// TIA Portal V17 export
// export: Created 2025-03-07T09:17:44.8534748Z, ExportSetting WithDefaults, DisplayName Totally Integrated Automation Portal, DisplayVersion V17 Update 8, DisplayName TIA Portal Openness, DisplayVersion V17 Update 8, DisplayName TIA Portal Version Control Interface, DisplayVersion V17, DisplayName SINAMICS Startdrive Advanced, DisplayVersion V17 SP2, DisplayName SINAMICS Startdrive G110M, G120, G120C, G120D, G120P, G115D, DisplayVersion V17 SP2, DisplayName SINAMICS Startdrive G130, G150, S120, S150, SINAMICS MV, S210, DisplayVersion V17 SP2, DisplayName STEP 7 Professional, DisplayVersion V17 Update 8, DisplayName SINUMERIK ONE STEP 7 Toolbox, DisplayVersion V17 Update 12, DisplayName SINUMERIK 840D sl STEP 7 Toolbox, DisplayVersion V17 Update 12, DisplayName STEP 7 Safety, DisplayVersion V17 Update 6, DisplayName WinCC Advanced, DisplayVersion V17 Update 8
DATA_BLOCK "DB2002_BA_MODES_MG1"   // DB2002
{ DB_Accessible_From_OPC_UA := 'FALSE' }
VERSION : 0.1
// stored: AutoNumber false, DBAccessibleFromOPCUA false, DBAccessibleFromWebserver true, InstanceOfName FB2002_BA_MODE, InstanceOfType FB
"FB2002_BA_MODE"
   // VAR_INPUT
   //    OPTIONS_0 { ExternalAccessible := 'False'; ExternalVisible := 'False'; ExternalWritable := 'False'} : Byte;
   //    BA1_BUTTON_I { ExternalAccessible := 'False'; ExternalVisible := 'False'; ExternalWritable := 'False'} : Bool;
   //    BA2_BUTTON_I { ExternalAccessible := 'False'; ExternalVisible := 'False'; ExternalWritable := 'False'} : Bool;
   //    BA3_BUTTON_I { ExternalAccessible := 'False'; ExternalVisible := 'False'; ExternalWritable := 'False'} : Bool;
   //    BA5_BUTTON_I { ExternalAccessible := 'False'; ExternalVisible := 'False'; ExternalWritable := 'False'} : Bool;
   //    SAFETY_ENABLED_W_DOOR_OPENED { ExternalAccessible := 'False'; ExternalVisible := 'False'; ExternalWritable := 'False'} : Bool;
   //    SAFETY_GATES_CLSD_AND_LCKD { ExternalAccessible := 'False'; ExternalVisible := 'False'; ExternalWritable := 'False'} : Bool;
   //    START_SERVICES_GLOBAL { ExternalAccessible := 'False'; ExternalVisible := 'False'; ExternalWritable := 'False'} : Bool;
   //    ANY_MCH_CYCLE_RUN { ExternalAccessible := 'False'; ExternalVisible := 'False'; ExternalWritable := 'False'} : Bool;
   //    MCH_RESET_FAULTS { ExternalAccessible := 'False'; ExternalVisible := 'False'; ExternalWritable := 'False'} : Bool;
   // END_VAR
   // VAR_OUTPUT
   //    NO_BA_MODE_SLCTD_WRN { ExternalAccessible := 'False'; ExternalVisible := 'False'; ExternalWritable := 'False'} : Bool;
   //    CHANGE_TO_BA1_MODE_WRN { ExternalAccessible := 'False'; ExternalVisible := 'False'; ExternalWritable := 'False'} : Bool;
   //    CHANGE_TO_BA2_MODE_WRN { ExternalAccessible := 'False'; ExternalVisible := 'False'; ExternalWritable := 'False'} : Bool;
   //    CHANGE_TO_BA3_MODE_WRN { ExternalAccessible := 'False'; ExternalVisible := 'False'; ExternalWritable := 'False'} : Bool;
   //    CHANGE_TO_BA5_MODE_WRN { ExternalAccessible := 'False'; ExternalVisible := 'False'; ExternalWritable := 'False'} : Bool;
   //    BA1_MODE_LED_O { ExternalAccessible := 'False'; ExternalVisible := 'False'; ExternalWritable := 'False'} : Bool;
   //    BA2_MODE_LED_O { ExternalAccessible := 'False'; ExternalVisible := 'False'; ExternalWritable := 'False'} : Bool;
   //    BA3_MODE_LED_O { ExternalAccessible := 'False'; ExternalVisible := 'False'; ExternalWritable := 'False'} : Bool;
   // END_VAR
   // VAR_IN_OUT
   //    MODE_GROUP_GENERAL_DB : "AUTO_SINGLE_SEMI_MANUAL";
   //    MODE_GROUP_BA_DB : "BA_MODE";
   // END_VAR
BEGIN
END_DATA_BLOCK
